# B&R Automation Studio project ARuser
Automation Studio 6.1.1.14; technology packages: mappView 6.1.1, OpcUaCs 6.0.0

## Configuration PC

CPU PC_any, AutomationRuntime 6.1.1, Build 11.3.0, Safety 0.0, Vc 

### Hardware
```
PC : PC_any v1.1.2.0 (OrderNumber=PC)
  Connector IF3:
    InaPort = 11159
  ConfigurationID = ARuser_PC
  VolatileGlobalPvSize = 200000
  Cyclic1Duration = 10000
  Cyclic3Tolerance = 60000000
  Cyclic8Duration = 10000
  FileDevice1
  FileDeviceName1 = FileDevice
  FileDevicePath1 = C:\Users\hendricksf\Desktop
  ActivateFtpServer = 1
  ActivateWebServer = 1
  ActivateSdm = 1
```

## Configuration X20CP

CPU X20CP3585, AutomationRuntime J4.93, Build 4.1.2, Vc V4.52.0

CPU X20CP3685, AutomationRuntime 6.1.1, Build 11.3.0, Vc 

### Hardware
```
X20CP3685 : X20CP3685 v1.8.1.0
  Connector IF2:
    ActivateDevice = 1
  Connector IF3:
    DNAConfiguration = manual
  ConfigurationID = ARuser_X20CP
  UserPartitionSize = 16
  VolatileGlobalPvSize = 120000
  FileDevice1
  FileDeviceName1 = USER
  FileDevicePath1 = USER_PATH
```

## Logical view

Binary libraries used (declarations not repeated): ArUser, MpUserX 5.24.3

### sys_lib.var
```iecst
(*error codes of the SYS_LIB services*)
VAR CONSTANT
	ERR_BUR_MO_NOTFOUND     	: UINT	:= 3019;    (*module not found*)
	ERR_BUR_ILLSTATE			: UINT	:= 3302;	(*illegal state of object*)
	ERR_BUR_ILLTYP				: UINT	:= 3311;	(*SYSreset - invalid input value for mode*)
	ERR_BUR_ILLPAR				: UINT	:= 3317;	(*illegal parameter*)
	ERR_BUR_ILLOBJ				: UINT	:= 3324;	(*object does not exist*)
	ERR_BUR_NOENTRY         	: UINT	:= 3332;    (*no entry*)
	ERR_BUR_TOOLONG_PVNAME		: UINT	:= 3333;	(*too long PV name*)
	ERR_BUR_ILLIDENT        	: UINT	:= 3336;    (*illegal ident*)
	ERR_BUR_NOTIME				: UINT	:= 3584;	(*time not available*)
	ERR_BUR_TMP_ALLOC			: UINT	:= 3601;	(*not enough continuous memory*)
	ERR_BUR_TMP_FREE			: UINT	:= 3701;	(*invalid pointer/length*)
END_VAR

(*state for object PLC task*)
VAR CONSTANT
	Z_ST_created				: UINT	:= 1;		(*object installed*)
	Z_ST_running				: UINT	:= 2;		(*object running*)
	Z_ST_blocked				: UINT	:= 3;		(*object stopped*)
	Z_ST_exist					: UINT	:= 16#00;	(*object exists*)
	Z_ST_installed				: UINT	:= 16#82;	(*temporary status during installation*)
	Z_ST_PVinstalled			: UINT	:= 16#83;	(*temporary status during installation*)
	Z_ST_IOinstalled			: UINT	:= 16#84;	(*temporary status during installation*)
	Z_ST_IOdeinstalled			: UINT	:= 16#85;	(*temporary status during installation*)
	Z_ST_PVdeinstalled			: UINT	:= 16#86;	(*temporary status during installation*)
	Z_ST_delete					: UINT	:= 16#87;	(*temporary status during installation*)
	Z_ST_stdebug				: UINT	:= 16#88;	(*temporary status during installation*)
	Z_ST_tmp_suspended			: UINT	:= 16#90;	(*object temporarily stopped*)
END_VAR

(*elementary data types*)
VAR CONSTANT
	SYSLIB_IEC_TYPE_USER_DEFINED	: USINT	:= 0;	(*User-defined data type*)
	SYSLIB_IEC_TYPE_USER_DEFINED_2	: USINT	:= 15;	(*User-defined data type (legacy: array of structs)*)
	SYSLIB_IEC_TYPE_BOOL			: USINT	:= 1;	(*8 Bit containing a boolean value FALSE=0 or TRUE=1*)
	SYSLIB_IEC_TYPE_SINT			: USINT	:= 2;	(*8 Bit signed integer*)
	SYSLIB_IEC_TYPE_INT				: USINT	:= 3;	(*16 Bit signed integer*)
	SYSLIB_IEC_TYPE_DINT			: USINT	:= 4;	(*32 Bit signed integer*)
	SYSLIB_IEC_TYPE_USINT			: USINT	:= 5;	(*8 Bit unsigned integer*)
	SYSLIB_IEC_TYPE_UINT			: USINT	:= 6;	(*16 Bit unsigned integer*)
	SYSLIB_IEC_TYPE_UDINT			: USINT	:= 7;	(*32 Bit unsigned integer*)
	SYSLIB_IEC_TYPE_REAL			: USINT	:= 8;	(*32 Bit floating point number*)
	SYSLIB_IEC_TYPE_STRING			: USINT	:= 9;	(*Variable-length single-byte character string*)
	SYSLIB_IEC_TYPE_DATE_AND_TIME	: USINT	:= 11;	(*32 Bit of Date in Seconds since 01.01.1970 00:00:00*)
	SYSLIB_IEC_TYPE_TIME			: USINT	:= 12;	(*32 Bit of Time in ms*)
	SYSLIB_IEC_TYPE_DATE			: USINT	:= 13;	(*32 Bit of Date (only)*)
	SYSLIB_IEC_TYPE_LREAL			: USINT	:= 14;	(*64 Bit floating point number*)
	SYSLIB_IEC_TYPE_TIME_OF_DAY		: USINT	:= 16;	(*32 Bit Time of day (only)*)
	SYSLIB_IEC_TYPE_BYTE			: USINT	:= 17;	(*Bit string of length 8*)
	SYSLIB_IEC_TYPE_WORD			: USINT	:= 18;	(*Bit string of length 16*)
	SYSLIB_IEC_TYPE_DWORD			: USINT	:= 19;	(*Bit string of length 32*)
	SYSLIB_IEC_TYPE_WSTRING			: USINT	:= 21;	(*Variable-length double-byte character string*)
END_VAR

(*shutdown/reboot types*)
VAR CONSTANT
	SYSLIB_WARMSTART				: USINT	:= 16#01;	(*WARMSTART (with restart)*)
	SYSLIB_COLDSTART				: USINT	:= 16#02;	(*COLDSTART (with restart)*)
	SYSLIB_WARMSTART_NO_REBOOT		: USINT	:= 16#11;	(*WARMSTART (no restart, only shutdown)*)
	SYSLIB_COLDSTART_NO_REBOOT		: USINT	:= 16#12;	(*COLDSTART (no restart, only shutdown)*)
	SYSLIB_DIAGNOSTICS				: USINT	:= 16#20;	(*DIAGNOSTICS (with restart)*)
	SYSLIB_SERVICE					: USINT	:= 16#40;	(*SERVICE (with restart) *)
END_VAR
```

### UserVariables.var
```iecst
(*Global constants*)
VAR CONSTANT
	MAX_USER_ROLES : USINT := 20; (*Maximum number of user roles*)
	MAX_USER_NAMES : USINT := 50; (*Maximum number of users*)
	MAX_USER_CLIENTS : USINT := 2; (*Maximum number of concurrent web clients*)
	MAX_USER_ITEM_LEN : USINT := 60; (*String length for users and roles*)
END_VAR
VAR
	DEFAULT_ROLE : STRING[80] := 'Everyone'; (*Default role when user was created*)
END_VAR
(*Global variable structure*)
VAR
	ArUser : userMAIN; (*Type for user data management*)
	RFID : rfidMAIN;
END_VAR
```

### changelog.txt
```
Version 1.2
- Update project to AS6
- Workaround for user create not assigning default role

Version 1.1
- Dont disable enable button in RFID group
- Added user partition for export/import
- Fixed export path not connected to ArUser.PAR.FilePath in mappView

Version 1.0
- Fixed password is not created

Version 0.8
- Update user management to version 0.8
- Added support for RFID reader 5E9030

Version 0.7
- Clear password field when user is created, password is changed, login or logout
- Removed user anonymous from user list
- Increased length of status message

Version 0.6
- Added message box before deleting user
- Changed constant to avoid conflict with other samples
- Fixed user selection after create and rename
- Updated mappView to 5.7.1
- Code optimizations

Version 0.5
- Code cleanup

Version 0.5
- Multi client support
- Changed error structure

Version 0.4
- Software structure change to work with future expansion
- Make sure passwords match before user is created
- Added support for RFID reader

Version 0.3
- Automatically set password when new user is created
- Erase password field when user logs out
- New command to rename user

Version 0.2
- Make sure last user can not be deleted
- Make sure last user can not delete himself
- Make sure last user can not be deleted
- Added group box with login
- Added message boxes for success and failed commands
- Visual tweaks and bugfixes

Version 0.1
- First public release
```

### Program Logical/mappUser/UserManagement

#### Variables.var
```iecst
(*General*)
VAR
	UserManagementState : userManagementEnum := IdleUser; (*State Machine for UserManagementState*)
	ArUserCreate_0 : ArUserCreate; (*Create an user with given name; default no password *)
	ArUserDelete_0 : ArUserDelete; (*Delete an user  *)
	ArUserExport_0 : ArUserExportEx; (*Export all user and role data*)
	ArUserImport_0 : ArUserImportEx; (*Import all user and role data*)
	ArUserSetPassword_0 : ArUserSetPassword; (*Set user password*)
	ArUserAssignRole_0 : ArUserAssignRole; (*Aisign a role to a user*)
	ArUserReleaseRole_0 : ArUserReleaseRole; (*Remove a role from a user*)
	ArUserGetNext_0 : ArUserGetNext; (*Get next user information*)
	ArUserGetFirst_0 : ArUserGetFirst; (*Get first user information*)
	ArUserInitList_0 : ArUserInitList; (*Initialize user or role list*)
	ArUserDestroyList_0 : ArUserDestroyList; (*Free up memory for list*)
	ArUserIdent : ArUserIdentType; (*Ident from user ot role list*)
	ArUserGetProperty_0 : ArUserGetProperty; (*Read property*)
	ArUserSetProperty_0 : ArUserSetProperty; (*Write a property*)
	PropertyName : STRING[100]; (*Name of the property*)
	tmpUserIdx : USINT;
	tmpUser : STRING[MAX_USER_ITEM_LEN];
	tmpUserOld : STRING[MAX_USER_ITEM_LEN];
	tmpUserNew : STRING[MAX_USER_ITEM_LEN];
	idx : USINT;
	idy : USINT;
	override : USINT;
END_VAR
VAR CONSTANT
	MAX_CYCLES : USINT := 10; (*Maximum number of override cycles*)
END_VAR
(*Loop counter*)
VAR
	RoleCounter : USINT;
	UserCounter : USINT;
	UserCounterTotal : ARRAY[0..MAX_USER_CLIENTS] OF USINT;
END_VAR
(*List types *)
VAR CONSTANT
	USER_LISTTYPE : BYTE := 1; (*List Type User*)
	ROLE_LISTTYPE : BYTE := 2; (*List Type Role*)
	USERROLE_LISTTYPE : BYTE := 3; (*List Type UserRole*)
END_VAR
(*Error Constants*)
VAR CONSTANT
	ERR_PASSWORD_MISMATCH : DINT := 50000; (*Passwords dont match*)
	ERR_USER_LIST_TOO_SHORT : DINT := 50001; (*More users found than fit into user list*)
	ERR_ROLE_LIST_TOO_SHORT : DINT := 50002; (*More roles found than fit into the role list*)
	ERR_DELETE_CURRENT_USER : DINT := 50003; (*Logged in user can not be deleted*)
	ERR_RENAME_CURRENT_USER : DINT := 50004; (*Logged in user can not be renamed*)
	ERR_USER_ROLE_NAME_SIZE : DINT := 50005; (*Logged in user can not be renamed*)
	ERR_USER_TOO_MANY_CLIENTS : DINT := 50010; (*More than 3 clients try to connect to user managment*)
	END_OF_LIST : DINT := -2144327714; (*End of list reached*)
	ONE : BOOL := TRUE;
END_VAR
```

#### Main.st
```iecst
// --------------------------------------------------------------------------------------------------------------------
// General user task. This is a support task for the mappView visualization. The following functions are implemneted
// - Create,rename and delete user
// - Create and delete roles
// - Change password and assign roles to users
// - Export and import user data
// Version 0.8
// --------------------------------------------------------------------------------------------------------------------
PROGRAM _INIT
	ArUser.CMD.ListRefresh	:= TRUE;								// Refresh user data on boot
END_PROGRAM

PROGRAM _CYCLIC

	FOR override:=0 TO MAX_CYCLES DO
		// --------------------------------------------------------------------------------------------------------------------
		// User managment state machine
		// --------------------------------------------------------------------------------------------------------------------
		CASE UserManagementState OF
			// --------------------------------------------------------------------------------------------------------------------
			// Wait for new command
			// --------------------------------------------------------------------------------------------------------------------
			IdleUser:
				// --------------------------------------------------------------------------------------------------------------------
				// Make sure we dont exceed maximum number of web clients
				IF(ArUser.PAR.VisuSlotID >= SIZEOF(ArUser.VIS)/SIZEOF(ArUser.VIS[0])) THEN
					ArUser.ERR.No := ERR_USER_TOO_MANY_CLIENTS;
					ArUser.ERR.State := UserManagementState;
					UserManagementState := ErrorUser;
					RETURN;
				END_IF

				// --------------------------------------------------------------------------------------------------------------------
				// Some general UI tasks
				FOR idy:=0 TO SIZEOF(ArUser.VIS)/SIZEOF(ArUser.VIS[0])-1 DO
					// --------------------------------------------------------------------------------------------------------------------
					// Create role list for current user
					idx := 0;
					brsmemset(ADR(ArUser.VIS[idy].ListUserRole), 0, SIZEOF(ArUser.VIS[idy].ListUserRole));
					WHILE brsstrcmp(ADR(ArUser.DAT.Users[ArUser.VIS[idy].ListUserIndex].Roles[idx]), ADR('')) <> 0 DO
						String2DataProvider(ADR(ArUser.DAT.Users[ArUser.VIS[idy].ListUserIndex].Roles[idx]), ADR(ArUser.VIS[idy].ListUserRole[idx]));
						idx := idx + 1;
					END_WHILE;
					// Make sure we dont delete last user role
					IF(idx > 1) THEN
						ArUser.VIS[idy].RoleDeleteEnabled := TRUE;
					ELSE
						ArUser.VIS[idy].RoleDeleteEnabled := FALSE;
					END_IF
					// Make sure we dont delete last user
					IF(UserCounterTotal[idy] > 0) THEN
						ArUser.VIS[idy].UserDeleteEnabled := TRUE;
					ELSE
						ArUser.VIS[idy].UserDeleteEnabled := FALSE;
					END_IF
				END_FOR;

				// --------------------------------------------------------------------------------------------------------------------
				// Create new user
				IF  (ArUser.CMD.UserCreate) THEN
					// Make sure passwords match before user is created
					IF((ArUser.PAR.Password <> '' OR ArUser.PAR.PasswordRepeat <> '') AND ArUser.PAR.Password <> ArUser.PAR.PasswordRepeat) THEN
						ArUser.ERR.No := ERR_PASSWORD_MISMATCH;
						ArUser.ERR.State := UserManagementState;
						UserManagementState := ErrorUser;
					ELSE
						tmpUser := ArUser.PAR.UserName;
						ArUserCreate_0(Execute := FALSE);
						ArUserSetPassword_0(Execute := FALSE);
						UserManagementState := CreateUser;
					END_IF
				// Assign role to user
				ELSIF (ArUser.CMD.RoleAssign) THEN
					tmpUser := ArUser.PAR.UserName;
					ArUserAssignRole_0(Execute := FALSE);
					ArUser.PAR.UserRole := ArUser.DAT.Roles[ArUser.VIS[ArUser.PAR.VisuSlotID].ListRoleIndex];
					UserManagementState := AssignRole;
				// Remove role from user
				ELSIF (ArUser.CMD.RoleRemove) THEN
					tmpUser := ArUser.PAR.UserName;
					ArUserReleaseRole_0(Execute := FALSE);
					ArUser.PAR.UserRole := ArUser.DAT.Users[ArUser.VIS[ArUser.PAR.VisuSlotID].ListUserIndex].Roles[ArUser.VIS[ArUser.PAR.VisuSlotID].ListUserRoleIndex];
					UserManagementState := ReleaseRole;
				// Delete user
				ELSIF (ArUser.CMD.UserDelete) THEN
					// Make sure we dont delete user that is logged in
					IF(brsstrcmp(ADR(ArUser.DAT.UserActive[ArUser.PAR.VisuSlotID]), ADR(ArUser.PAR.UserName)) = 0) THEN
						ArUser.ERR.No := ERR_DELETE_CURRENT_USER;
						ArUser.ERR.State := UserManagementState;
						UserManagementState := ErrorUser;
					ELSE
						tmpUser := ArUser.PAR.UserName;
						ArUserDelete_0(Execute := FALSE);
						UserManagementState := DeleteUser;
					END_IF
				// Rename user
				ELSIF (ArUser.CMD.UserRename) THEN
					// Make sure we dont delete user that is logged in
					IF(brsstrcmp(ADR(ArUser.DAT.UserActive[ArUser.PAR.VisuSlotID]), ADR(ArUser.PAR.UserName)) = 0) THEN
						ArUser.ERR.No := ERR_RENAME_CURRENT_USER;
						ArUser.ERR.State := UserManagementState;
						UserManagementState := ErrorUser;
					ELSE
						tmpUserOld := ArUser.PAR.UserName;
						tmpUser := ArUser.PAR.UserNameNew;
						ArUserGetProperty_0(Execute := FALSE);
						ArUserSetProperty_0(Execute := FALSE);
						ArUserAssignRole_0(Execute := FALSE);
						ArUserDelete_0(Execute := FALSE);
						UserManagementState := RenameUser;
					END_IF
				// Export user data
				ELSIF (ArUser.CMD.Export) THEN
					ArUserExport_0(Execute := FALSE);
					UserManagementState := ExportList;
				// Import user data
				ELSIF (ArUser.CMD.Import) THEN
					ArUserImport_0(Execute := FALSE);
					UserManagementState := ImportList;
				// Change user password
				ELSIF (ArUser.CMD.PasswordChange) THEN
					tmpUser := ArUser.PAR.UserName;
					ArUserSetPassword_0(Execute := FALSE);
					UserManagementState := ComparePassword;
				// Refresh user list
				ELSIF (ArUser.CMD.ListRefresh) THEN
					tmpUser := '';
					UserManagementState := CreateUserListGetFirst;
				END_IF;

				// --------------------------------------------------------------------------------------------------------------------
				// Reset fields on new command
				FOR idx:=0 TO SIZEOF(ArUser.CMD) DO
					IF brsmemcmp(ADR(ArUser.CMD) + idx, ADR(ONE), 1) = 0 THEN
						ArUser.DAT.Status := '';
	 				END_IF
				END_FOR
				ArUser.CMD.ErrorReset := FALSE;

				// Abot override when no command is active
				IF (UserManagementState = IdleUser) THEN
					RETURN;
				END_IF
			// --------------------------------------------------------------------------------------------------------------------
			// Create new user
			// --------------------------------------------------------------------------------------------------------------------
			CreateUser:
				ArUserCreate_0(Execute := TRUE , UserName := tmpUser);

				// --------------------------------------------------------------------------------------------------------------------
				// Success
				IF ArUserCreate_0.Done AND NOT ArUserCreate_0.Busy THEN
					// Create new user
					IF(ArUser.CMD.UserCreate) THEN
						// --------------------------------------------------------------------------------------------------------------------
						// Success
						ArUserAssignRole_0(Execute := TRUE, UserName := tmpUser, RoleName := DEFAULT_ROLE);
						ArUserAssignRole_0(Execute := TRUE, UserName := tmpUser, RoleName := DEFAULT_ROLE);
						IF ArUserAssignRole_0.Done AND NOT ArUserAssignRole_0.Busy THEN
							ArUserAssignRole_0(Execute := FALSE);

							ArUser.DAT.Status := 'User ';
							brsstrcat(ADR(ArUser.DAT.Status), ADR(tmpUser));
							brsstrcat(ADR(ArUser.DAT.Status), ADR(' created'));
							// Set password when it exists
							IF ArUser.PAR.Password <> '' THEN
								UserManagementState := ComparePassword;
							ELSE
								ArUser.PAR.UserName := '';
								UserManagementState := CreateUserListGetFirst;
							END_IF;

							RETURN;
							// Error
						ELSIF ArUserAssignRole_0.Error THEN
							ArUser.ERR.No := ArUserAssignRole_0.ErrorID;
							ArUser.ERR.State := UserManagementState;
							UserManagementState := ErrorUser;
						END_IF
						// Rename existing user
					ELSE
						PropertyName := 'UserID';
						UserManagementState := PropertyRead;
					END_IF
					// Error
				ELSIF ArUserCreate_0.Error THEN
					ArUser.ERR.No := ArUserCreate_0.ErrorID;
					ArUser.ERR.State := UserManagementState;
					UserManagementState := ErrorUser;
				END_IF;

			// --------------------------------------------------------------------------------------------------------------------
			// Assign user role
			// --------------------------------------------------------------------------------------------------------------------
			AssignRole:
				ArUserAssignRole_0(Execute := TRUE, UserName := tmpUser, RoleName := ArUser.PAR.UserRole);

				// --------------------------------------------------------------------------------------------------------------------
				// Success
				IF ArUser.CMD.RoleAssign AND ArUserAssignRole_0.Done AND NOT ArUserAssignRole_0.Busy THEN
					ArUser.DAT.Status := 'Role >';
					brsstrcat(ADR(ArUser.DAT.Status), ADR(ArUser.PAR.UserRole));
					brsstrcat(ADR(ArUser.DAT.Status), ADR('< assigned to user '));
					brsstrcat(ADR(ArUser.DAT.Status), ADR(tmpUser));
					ArUser.PAR.UserName := '';
					UserManagementState := CreateUserListGetFirst;
				ELSIF ArUser.CMD.UserRename AND ((ArUserAssignRole_0.Done AND NOT ArUserAssignRole_0.Busy) OR (ArUserAssignRole_0.ErrorID = arUSER_ERR_ALREADY_EXISTS)) THEN
					idx := idx +1;
					// Assign next role if it exists
					IF ArUser.DAT.Users[tmpUserIdx].Roles[idx] <> '' AND idx < MAX_USER_ROLES THEN
						ArUserAssignRole_0(Execute := FALSE);
						ArUser.PAR.UserRole := ArUser.DAT.Users[tmpUserIdx].Roles[idx];
					// Delete old user
					ELSE
						// Move user names around
						tmpUserNew 	:= tmpUser;
						tmpUser 	:= tmpUserOld;
						UserManagementState := DeleteUser;
					END_IF
				// Error
				ELSIF ArUserAssignRole_0.Error THEN
					ArUser.ERR.No := ArUserAssignRole_0.ErrorID;
					ArUser.ERR.State := UserManagementState;
					UserManagementState := ErrorUser;
				END_IF;

			// --------------------------------------------------------------------------------------------------------------------
			// Release user role
			// --------------------------------------------------------------------------------------------------------------------
			ReleaseRole:
				ArUserReleaseRole_0(Execute := TRUE, UserName := tmpUser, RoleName := ArUser.PAR.UserRole);

				// --------------------------------------------------------------------------------------------------------------------
				// Success
				IF ArUserReleaseRole_0.Done AND NOT ArUserReleaseRole_0.Busy THEN
					ArUser.DAT.Status := 'Role >';
					brsstrcat(ADR(ArUser.DAT.Status), ADR(ArUser.PAR.UserRole));
					brsstrcat(ADR(ArUser.DAT.Status), ADR('< removed from user '));
					brsstrcat(ADR(ArUser.DAT.Status), ADR(tmpUser));
					ArUser.PAR.UserName := '';
					UserManagementState := CreateUserListGetFirst;
				// Error
				ELSIF ArUserReleaseRole_0.Error THEN
					ArUser.ERR.No := ArUserReleaseRole_0.ErrorID;
					ArUser.ERR.State := UserManagementState;
					UserManagementState := ErrorUser;
				END_IF;

			// --------------------------------------------------------------------------------------------------------------------
			// Delete user
			// --------------------------------------------------------------------------------------------------------------------
			DeleteUser:
				ArUserDelete_0(Execute := TRUE, UserName := tmpUser);

				// --------------------------------------------------------------------------------------------------------------------
				// Success
				IF ArUserDelete_0.Done AND NOT ArUserDelete_0.Busy THEN
					// User delete command
					IF ArUser.CMD.UserDelete THEN
						ArUser.DAT.Status := 'User >';
						brsstrcat(ADR(ArUser.DAT.Status), ADR(tmpUser));
						brsstrcat(ADR(ArUser.DAT.Status), ADR('< deleted'));
						// User rename command
					ELSE
						ArUser.DAT.Status := 'User ';
						brsstrcat(ADR(ArUser.DAT.Status), ADR(tmpUserOld));
						brsstrcat(ADR(ArUser.DAT.Status), ADR(' renamed to >'));
						brsstrcat(ADR(ArUser.DAT.Status), ADR(ArUser.PAR.UserNameNew));
						brsstrcat(ADR(ArUser.DAT.Status), ADR('<'));
					END_IF
					ArUser.PAR.UserName := '';
					tmpUser := '';
					UserManagementState := CreateUserListGetFirst;
				// Error
				ELSIF ArUserDelete_0.Error THEN
					ArUser.ERR.No := ArUserDelete_0.ErrorID;
					ArUser.ERR.State := UserManagementState;
					UserManagementState := ErrorUser;
				END_IF;

			// --------------------------------------------------------------------------------------------------------------------
			// Rename user
			// --------------------------------------------------------------------------------------------------------------------
			RenameUser:
				tmpUserIdx := 0;
				// Find user name in list
				WHILE (brsstrcmp(ADR(ArUser.DAT.Users[tmpUserIdx].Name), ADR(tmpUserOld)) <> 0) AND (tmpUserIdx < MAX_USER_NAMES) DO
					tmpUserIdx := tmpUserIdx + 1;
				END_WHILE;

				// --------------------------------------------------------------------------------------------------------------------
				// Success
				IF(tmpUserIdx < MAX_USER_NAMES) THEN
					ArUserCreate_0(Execute := FALSE);
					UserManagementState := CreateUser;
				// Error when user was not found
				ELSE
					ArUser.ERR.No := arUSER_ERR_DOES_NOT_EXIST;
					ArUser.ERR.State := UserManagementState;
					UserManagementState := ErrorUser;
				END_IF

			// --------------------------------------------------------------------------------------------------------------------
			// Read user property
			// --------------------------------------------------------------------------------------------------------------------
			PropertyRead:
				ArUserGetProperty_0(Execute := TRUE, ElementType := arUSER_USER_PROPERTIES, ElementName := tmpUserOld, PropertyName := PropertyName);

				// --------------------------------------------------------------------------------------------------------------------
				// Success
				IF ArUserGetProperty_0.Done AND NOT ArUserGetProperty_0.Busy THEN
					ArUserSetProperty_0(Execute := FALSE);
					UserManagementState := PropertyWrite;
				// Error
				ELSIF ArUserGetProperty_0.Error THEN
					ArUser.ERR.No := ArUserGetProperty_0.ErrorID;
					ArUser.ERR.State := UserManagementState;
					UserManagementState := ErrorUser;
				END_IF;
			// --------------------------------------------------------------------------------------------------------------------
			// Write user property
			// --------------------------------------------------------------------------------------------------------------------
			PropertyWrite:
				ArUserSetProperty_0(Execute := TRUE, ElementType := arUSER_USER_PROPERTIES, ElementName := tmpUser, PropertyName := PropertyName, PropertyValue := ArUserGetProperty_0.PropertyValue);

				// --------------------------------------------------------------------------------------------------------------------
				// Success
				IF ArUserSetProperty_0.Done AND NOT ArUserSetProperty_0.Busy THEN
					// Read password after user ID
					IF PropertyName = 'UserID' THEN
						PropertyName := 'Password';
						ArUserGetProperty_0(Execute := FALSE);
						UserManagementState := PropertyRead;
						// Assign roles after password
					ELSIF PropertyName = 'Password' THEN
						idx := 0;
						ArUser.PAR.UserRole := ArUser.DAT.Users[tmpUserIdx].Roles[idx];
						UserManagementState := AssignRole;
					END_IF
				// Error
				ELSIF ArUserSetProperty_0.Error THEN
					ArUser.ERR.No := ArUserSetProperty_0.ErrorID;
					ArUser.ERR.State := UserManagementState;
					UserManagementState := ErrorUser;
				END_IF;

			// --------------------------------------------------------------------------------------------------------------------
			// Export user list to file
			// --------------------------------------------------------------------------------------------------------------------
			ExportList:
				ArUserExport_0(Execute := TRUE , LocalPath := ArUser.PAR.FilePath);

				// --------------------------------------------------------------------------------------------------------------------
				// Success
				IF ArUserExport_0.Done AND NOT ArUserExport_0.Busy THEN
					ArUser.DAT.Status := 'Export finished';
					ArUser.CMD.Export := FALSE;
					ArUser.VIS[ArUser.PAR.VisuSlotID].ShowMessageBoxOK := TRUE;
					UserManagementState := IdleUser;
					RETURN;
				// Error
				ELSIF ArUserExport_0.Error THEN
					ArUser.ERR.No := ArUserExport_0.ErrorID;
					ArUser.ERR.State := UserManagementState;
					UserManagementState := ErrorUser;
				END_IF;

			// --------------------------------------------------------------------------------------------------------------------
			// Import user list from file
			// --------------------------------------------------------------------------------------------------------------------
			ImportList:
				ArUserImport_0(Execute := TRUE , LocalPath := ArUser.PAR.FilePath);

				// --------------------------------------------------------------------------------------------------------------------
				// Success
				IF ArUserImport_0.Done AND NOT ArUserImport_0.Busy THEN
					ArUser.DAT.Status := 'Import finished';
					ArUser.CMD.Import := FALSE;
					ArUser.VIS[ArUser.PAR.VisuSlotID].ShowMessageBoxOK := TRUE;
					UserManagementState := CreateUserListGetFirst;
				// Error
				ELSIF ArUserImport_0.Error THEN
					ArUser.ERR.No := ArUserImport_0.ErrorID;
					ArUser.ERR.State := UserManagementState;
					UserManagementState := ErrorUser;
				END_IF;

			// --------------------------------------------------------------------------------------------------------------------
			// Change password, make sure both passwords are correct
			// --------------------------------------------------------------------------------------------------------------------
			ComparePassword:
				// --------------------------------------------------------------------------------------------------------------------
				// Success
				IF brsstrcmp(ADR(ArUser.PAR.Password), ADR(ArUser.PAR.PasswordRepeat)) = 0 THEN
					UserManagementState := ChangePassword;
				// Error
				ELSE
					ArUser.ERR.No := ERR_PASSWORD_MISMATCH;
					ArUser.ERR.State := UserManagementState;
					UserManagementState := ErrorUser;
				END_IF;

			// --------------------------------------------------------------------------------------------------------------------
			// Change password, execute password change
			// --------------------------------------------------------------------------------------------------------------------
			ChangePassword:
				ArUserSetPassword_0(Execute := TRUE, UserName := tmpUser, Password := ArUser.PAR.Password);

				// --------------------------------------------------------------------------------------------------------------------
				// Success
				IF ArUserSetPassword_0.Done AND NOT ArUserSetPassword_0.Busy THEN
					IF ArUser.CMD.PasswordChange THEN
						ArUser.DAT.Status := 'Password for user >';
						brsstrcat(ADR(ArUser.DAT.Status), ADR(tmpUser));
						brsstrcat(ADR(ArUser.DAT.Status), ADR('< changed'));
						ArUser.PAR.Password := '';
						ArUser.PAR.PasswordRepeat := '';
						ArUser.CMD.PasswordChange := FALSE;
						ArUser.VIS[ArUser.PAR.VisuSlotID].ShowMessageBoxOK := TRUE;
						UserManagementState := IdleUser;
						RETURN;
					ELSE
						UserManagementState := CreateUserListGetFirst;
					END_IF;
				// Error
				ELSIF ArUserSetPassword_0.Error THEN
					ArUser.ERR.No := ArUserSetPassword_0.ErrorID;
					ArUser.ERR.State := UserManagementState;
					UserManagementState := ErrorUser;
				END_IF;

			// --------------------------------------------------------------------------------------------------------------------
			// Create list of users and roles
			// --------------------------------------------------------------------------------------------------------------------
			CreateUserListGetFirst:
				// Initialize user list
				ArUserInitList_0(Execute := TRUE, ListType := USER_LISTTYPE, ElementName :='');

				// --------------------------------------------------------------------------------------------------------------------
				// Get first user name
				IF ArUserInitList_0.Done AND NOT ArUserInitList_0.Busy THEN
					ArUserGetFirst_0(Execute := TRUE , List := ArUserInitList_0.List );

					// --------------------------------------------------------------------------------------------------------------------
					// Success
					IF ArUserGetFirst_0.Done THEN
						// Clear data, store user name and generate data provider for vis
						brsmemset(ADR(ArUser.DAT.Users), 0, SIZEOF(ArUser.DAT.Users));
						brsmemset(ADR(ArUser.VIS[ArUser.PAR.VisuSlotID].ListUsers), 0, SIZEOF(ArUser.VIS[ArUser.PAR.VisuSlotID].ListUsers));
						brsmemset(ADR(ArUser.VIS[ArUser.PAR.VisuSlotID].ListRoles), 0, SIZEOF(ArUser.VIS[ArUser.PAR.VisuSlotID].ListRoles));
						UserCounter := 0;

						// Make sure user name fits
						IF(brsstrlen(ADR(ArUserGetFirst_0.ElementName)) < MAX_USER_ITEM_LEN) THEN
							// Ignore use an anonymous
							IF(ArUserGetFirst_0.ElementName <> 'Anonymous') THEN
								ArUser.DAT.Users[UserCounter].Name := ArUserGetFirst_0.ElementName;
								String2DataProvider(ADR(ArUserGetFirst_0.ElementName), ADR(ArUser.VIS[ArUser.PAR.VisuSlotID].ListUsers[UserCounter]));
								UserCounter := 1;
							ELSE
								UserCounter := 0;
							END_IF
							// Reset function block and init counters
							ArUserGetFirst_0(Execute := FALSE);
							RoleCounter := 0;
							UserManagementState := CreateUserListGetNext;
						// User name is too long
						ELSE
							ArUser.ERR.No := ERR_USER_ROLE_NAME_SIZE;
							ArUser.ERR.State := UserManagementState;
							UserManagementState := ErrorUser;
						END_IF;
					// Error
					ELSIF ArUserGetFirst_0.Error THEN
						ArUser.ERR.No := ArUserGetFirst_0.ErrorID;
						ArUser.ERR.State := UserManagementState;
						UserManagementState := ErrorUser;
					END_IF;
				// Error
				ELSIF ArUserInitList_0.Error THEN
					ArUser.ERR.No := ArUserInitList_0.ErrorID;
					ArUser.ERR.State := UserManagementState;
					UserManagementState := ErrorUser;
				END_IF;

			CreateUserListGetNext:
				// Make sure we have space left
				IF UserCounter < SIZEOF(ArUser.DAT.Users)/SIZEOF(ArUser.DAT.Users[0]) THEN
					// Get next user
					ArUserGetNext_0(Execute := TRUE , List := ArUserInitList_0.List);

					// --------------------------------------------------------------------------------------------------------------------
					// Success
					IF ArUserGetNext_0.Done THEN
						// Make sure user name fits
						IF(brsstrlen(ADR(ArUserGetNext_0.ElementName)) < MAX_USER_ITEM_LEN) THEN
							// Ignore use an anonymous
							IF(ArUserGetNext_0.ElementName <> 'Anonymous') THEN
								// Store user name and generate data provider for vis
								ArUser.DAT.Users[UserCounter].Name := ArUserGetNext_0.ElementName;
								String2DataProvider(ADR(ArUserGetNext_0.ElementName), ADR(ArUser.VIS[ArUser.PAR.VisuSlotID].ListUsers[UserCounter]));
								// Reset function block and get next name
								UserCounter := UserCounter + 1;
							END_IF
							ArUserGetNext_0(Execute := FALSE);
						// User name is too long
						ELSE
							ArUser.ERR.No := ERR_USER_ROLE_NAME_SIZE;
							ArUser.ERR.State := UserManagementState;
							UserManagementState := ErrorUser;
						END_IF;
					// Error
					ELSIF ArUserGetNext_0.Error AND NOT (ArUserGetNext_0.ErrorID = END_OF_LIST) THEN
						ArUser.ERR.No := ArUserGetNext_0.ErrorID;
						ArUser.ERR.State := UserManagementState;
						UserManagementState := ErrorUser;
					// List is complete
					ELSIF ArUserGetNext_0.ErrorID = END_OF_LIST THEN
						// Free up memory
						ArUserIdent := ArUserInitList_0.List;
						ArUserDestroyList_0(Execute := TRUE, List := ArUserIdent);
						ArUserDestroyList_0(Execute := FALSE, List := ArUserIdent);
						// Reset function blocks and counters
						ArUserGetNext_0(Execute := FALSE);
						ArUserGetFirst_0(Execute := FALSE);
						ArUserInitList_0(Execute := FALSE);
						UserCounterTotal[ArUser.PAR.VisuSlotID] := UserCounter;
						UserCounter := 0;
						RoleCounter := 0;
						UserManagementState := RoleListInitList;
					END_IF;
				// User list is too short
				ELSE
					ArUser.ERR.No := ERR_USER_LIST_TOO_SHORT;
					ArUser.ERR.State := UserManagementState;
					UserManagementState := ErrorUser;
				END_IF;

			// --------------------------------------------------------------------------------------------------------------------
			// Create table of roles assigned to the table of users
			// --------------------------------------------------------------------------------------------------------------------
			RoleListInitList:
				IF ArUser.DAT.Users[UserCounter].Name <> '' THEN
					ArUserInitList_0(Execute := TRUE, ListType := USERROLE_LISTTYPE , ElementName := ArUser.DAT.Users[UserCounter].Name);

					// --------------------------------------------------------------------------------------------------------------------
					// Success
					IF ArUserInitList_0.Done  AND NOT ArUserInitList_0.Busy THEN
						ArUserGetFirst_0(Execute := TRUE , List := ArUserInitList_0.List);
						// --------------------------------------------------------------------------------------------------------------------
						// Success
						IF ArUserGetFirst_0.Done THEN
							// Make sure role name fits
							IF(brsstrlen(ADR(ArUserInitList_0.ElementName)) < MAX_USER_ITEM_LEN) THEN
								ArUser.DAT.Users[UserCounter].Roles[0] := ArUserGetFirst_0.ElementName;
								ArUserGetFirst_0(Execute := FALSE , List := ArUserInitList_0.List);
								RoleCounter := 1;
								UserManagementState:= RoleListGetNext;
								// User role is too long
							ELSE
								ArUser.ERR.No := ERR_USER_ROLE_NAME_SIZE;
								ArUser.ERR.State := UserManagementState;
								UserManagementState := ErrorUser;
							END_IF;
						// Error
						ELSIF ArUserGetFirst_0.Error THEN
							ArUser.ERR.No := ArUserGetFirst_0.ErrorID;
							ArUser.ERR.State := UserManagementState;
							UserManagementState := ErrorUser;
						END_IF;
					// Error
					ELSIF ArUserInitList_0.Error THEN
						ArUser.ERR.No := ArUserInitList_0.ErrorID;
						ArUser.ERR.State := UserManagementState;
						UserManagementState := ErrorUser;
					END_IF;
				// Finish when user roles are complete
				ELSE
					// Reset function blocks
					ArUserInitList_0(Execute := FALSE);
					ArUserGetFirst_0(Execute := FALSE);
					UserCounter := 1;
					RoleCounter := 0;
					UserManagementState := CreateRoleListGetFirst;
				END_IF;

			RoleListGetNext:
				ArUserGetNext_0(Execute := TRUE, List := ArUserInitList_0.List);

				// --------------------------------------------------------------------------------------------------------------------
				// Success
				IF ArUserGetNext_0.Done THEN
					// Make sure user name fits
					IF(brsstrlen(ADR(ArUserGetNext_0.ElementName)) < MAX_USER_ITEM_LEN) THEN
						ArUser.DAT.Users[UserCounter].Roles[RoleCounter] := ArUserGetNext_0.ElementName;
						RoleCounter := RoleCounter + 1;
						ArUserGetNext_0(Execute := FALSE, List := ArUserInitList_0.List);
					// User role is too long
					ELSE
						ArUser.ERR.No := ERR_USER_ROLE_NAME_SIZE;
						ArUser.ERR.State := UserManagementState;
						UserManagementState := ErrorUser;
					END_IF;
				// List is complete
				ELSIF ArUserGetNext_0.ErrorID = END_OF_LIST THEN
					UserCounter := UserCounter + 1;
					// Free up memory
					ArUserIdent := ArUserInitList_0.List;
					ArUserDestroyList_0(Execute := TRUE, List := ArUserIdent);
					ArUserDestroyList_0(Execute := FALSE, List := ArUserIdent);
					// Reset function blocks
					ArUserGetNext_0(Execute := FALSE);
					ArUserInitList_0(Execute := FALSE);
					UserManagementState := RoleListInitList;
				// Error
				ELSIF ArUserGetNext_0.Error THEN
					ArUser.ERR.No := ArUserGetNext_0.ErrorID;
					ArUser.ERR.State := UserManagementState;
					UserManagementState := ErrorUser;
				END_IF;

			// --------------------------------------------------------------------------------------------------------------------
			// Create table of roles
			// --------------------------------------------------------------------------------------------------------------------
			CreateRoleListGetFirst:
				ArUserInitList_0(Execute := TRUE, ListType := ROLE_LISTTYPE , ElementName :='' );

				// --------------------------------------------------------------------------------------------------------------------
				// Success
				IF ArUserInitList_0.Done AND NOT ArUserInitList_0.Busy THEN
					ArUserGetFirst_0(Execute := TRUE , List := ArUserInitList_0.List );

					// --------------------------------------------------------------------------------------------------------------------
					// Store role names and generate data provider for vis
					IF ArUserGetFirst_0.Done THEN
						// Make sure role name fits
						IF(brsstrlen(ADR(ArUserGetFirst_0.ElementName)) < MAX_USER_ITEM_LEN) THEN
							ArUser.DAT.Roles[RoleCounter] := ArUserGetFirst_0.ElementName;
							String2DataProvider(ADR(ArUserGetFirst_0.ElementName), ADR(ArUser.VIS[ArUser.PAR.VisuSlotID].ListRoles[RoleCounter]));
							// Reset function block and init counters
							ArUserGetFirst_0(Execute := FALSE);
							RoleCounter := 1;
							UserManagementState := CreateRoleListGetNext;
							// Role name is too long
						ELSE
							ArUser.ERR.No := ERR_USER_ROLE_NAME_SIZE;
							ArUser.ERR.State := UserManagementState;
							UserManagementState := ErrorUser;
						END_IF;
					// Error
					ELSIF ArUserGetFirst_0.Error THEN
						ArUser.ERR.No := ArUserGetFirst_0.ErrorID;
						ArUser.ERR.State := UserManagementState;
						UserManagementState := ErrorUser;
					END_IF;
				// Error
				ELSIF ArUserInitList_0.Error THEN
					ArUser.ERR.No := ArUserInitList_0.ErrorID;
					ArUser.ERR.State := UserManagementState;
					UserManagementState := ErrorUser;
				END_IF;

			CreateRoleListGetNext:
				IF UserCounter < SIZEOF(ArUser.DAT.Roles)/SIZEOF(ArUser.DAT.Roles[0]) THEN
					ArUserGetNext_0(Execute := TRUE , List := ArUserInitList_0.List);

					// --------------------------------------------------------------------------------------------------------------------
					// Store user name and generate data provider for vis
					IF ArUserGetNext_0.Done THEN
						// Make sure user name fits
						IF(brsstrlen(ADR(ArUserGetNext_0.ElementName)) < MAX_USER_ITEM_LEN) THEN
							ArUser.DAT.Roles[RoleCounter] := ArUserGetNext_0.ElementName;
							String2DataProvider(ADR(ArUserGetNext_0.ElementName), ADR(ArUser.VIS[ArUser.PAR.VisuSlotID].ListRoles[RoleCounter]));
							// Reset function block and get next name
							RoleCounter := RoleCounter + 1;
							ArUserGetNext_0(Execute := FALSE);
						// Role name is too long
						ELSE
							ArUser.ERR.No := ERR_USER_ROLE_NAME_SIZE;
							ArUser.ERR.State := UserManagementState;
							UserManagementState := ErrorUser;
						END_IF;
					// Error
					ELSIF ArUserGetNext_0.Error AND NOT (ArUserGetNext_0.ErrorID = END_OF_LIST) THEN
						ArUser.ERR.No := ArUserGetNext_0.ErrorID;
						ArUser.ERR.State := UserManagementState;
						UserManagementState := ErrorUser;
					// End of list reached
					ELSIF ArUserGetNext_0.ErrorID = END_OF_LIST THEN
						// Show message box after succesful command except refresh
						IF(NOT ArUser.CMD.ListRefresh) THEN
							ArUser.VIS[ArUser.PAR.VisuSlotID].ShowMessageBoxOK := TRUE;
						END_IF
						// Reset function blocks
						ArUserGetNext_0(Execute := FALSE);
						ArUserInitList_0(Execute := FALSE);
						// Reset function blocks
						ArUserGetNext_0(Execute := FALSE);
						ArUserGetFirst_0(Execute := FALSE);
						ArUserInitList_0(Execute := FALSE);
						RoleCounter := 0;
						// Reset command
						brsmemset(ADR(ArUser.CMD), 0, SIZEOF(ArUser.CMD));
						// Select last user if possible
						IF(tmpUser <> '') THEN
							ArUser.VIS[ArUser.PAR.VisuSlotID].ListUserValue := tmpUser;
						ELSIF(tmpUserNew <> '') THEN
							ArUser.VIS[ArUser.PAR.VisuSlotID].ListUserValue := tmpUserNew;
						ELSE
							ArUser.PAR.UserName := ArUser.DAT.Users[0].Name;
						END_IF
						// Copy user data into all slots on first boot
						FOR idy:=0 TO SIZEOF(ArUser.VIS)/SIZEOF(ArUser.VIS[0])-1 DO
							IF(idy <> ArUser.PAR.VisuSlotID) THEN
								brsmemcpy(ADR(ArUser.VIS[idy].ListUsers), ADR(ArUser.VIS[ArUser.PAR.VisuSlotID].ListUsers), SIZEOF(ArUser.VIS[ArUser.PAR.VisuSlotID].ListUsers));
								brsmemcpy(ADR(ArUser.VIS[idy].ListRoles), ADR(ArUser.VIS[ArUser.PAR.VisuSlotID].ListRoles), SIZEOF(ArUser.VIS[ArUser.PAR.VisuSlotID].ListRoles));
								UserCounterTotal[idy] := UserCounterTotal[ArUser.PAR.VisuSlotID];
							END_IF
						END_FOR
						UserManagementState := IdleUser;
						RETURN;
					END_IF;
				// Role list is too short
				ELSE
					ArUser.ERR.No := ERR_ROLE_LIST_TOO_SHORT;
					ArUser.ERR.State := UserManagementState;
					UserManagementState := ErrorUser;
				END_IF;

			// --------------------------------------------------------------------------------------------------------------------
			// Error
			// --------------------------------------------------------------------------------------------------------------------
			ErrorUser:
				// --------------------------------------------------------------------------------------------------------------------
				// Reset function blocks
				ArUserInitList_0(Execute := FALSE);
				ArUserGetFirst_0(Execute := FALSE);
				ArUserGetNext_0(Execute := FALSE);
				ArUserCreate_0(Execute := FALSE);
				ArUserReleaseRole_0(Execute := FALSE);
				ArUserReleaseRole_0(Execute := FALSE);
				ArUserDelete_0(Execute := FALSE);
				ArUserGetProperty_0(Execute := FALSE);
				ArUserSetProperty_0(Execute := FALSE);
				ArUserSetPassword_0(Execute := FALSE);
				ArUserImport_0(Execute := FALSE);
				ArUserExport_0(Execute := FALSE);

				// --------------------------------------------------------------------------------------------------------------------
				// Generate text for most common errors
				IF(ArUser.ERR.No = arUSER_ERR_ALREADY_EXISTS) THEN
					ArUser.ERR.Text := 'ERR: User/Role already exists or is already assigned';
				ELSIF(ArUser.ERR.No = arUSER_ERR_PARAMETER) THEN
					ArUser.ERR.Text := 'ERR: User/Role is empty';
				ELSIF(ArUser.ERR.No = arUSER_ERR_DOES_NOT_EXIST) THEN
					ArUser.ERR.Text := 'ERR: User/Role does not exist';
				ELSIF(ArUser.ERR.No = ERR_PASSWORD_MISMATCH) THEN
					ArUser.ERR.Text := 'ERR: Passwords do not match';
				ELSIF(ArUser.ERR.No = ERR_USER_LIST_TOO_SHORT) THEN
					ArUser.ERR.Text := 'ERR: User list is too short';
				ELSIF(ArUser.ERR.No = ERR_ROLE_LIST_TOO_SHORT) THEN
					ArUser.ERR.Text := 'ERR: Role list is too short';
				ELSIF(ArUser.ERR.No = ERR_DELETE_CURRENT_USER) THEN
					ArUser.ERR.Text := 'ERR: Can not delete user that is logged in';
				ELSIF(ArUser.ERR.No = ERR_USER_ROLE_NAME_SIZE) THEN
					ArUser.ERR.Text := 'ERR: User name or role exceeds maximum size of ITEM_LENGTH';
				ELSIF(ArUser.ERR.No = ERR_RENAME_CURRENT_USER) THEN
					ArUser.ERR.Text := 'ERR: Can not rename user that is logged in';
				ELSE
					ArUser.ERR.Text := 'Error executing command';
				END_IF
				// Make sure we dont exceed maximum number of web clients
				IF(ArUser.PAR.VisuSlotID < SIZEOF(ArUser.VIS)/SIZEOF(ArUser.VIS[0])) THEN
					ArUser.VIS[ArUser.PAR.VisuSlotID].ShowMessageBoxError := TRUE;
				END_IF
				// --------------------------------------------------------------------------------------------------------------------
				// Return to idle state
				IF ArUser.CMD.ErrorReset THEN
					UserCounter := 1;
					RoleCounter := 0;

					brsmemset(ADR(ArUser.ERR), 0, SIZEOF(ArUser.ERR));
					ArUser.CMD.ErrorReset := FALSE;
					ArUser.VIS[ArUser.PAR.VisuSlotID].ShowMessageBoxError := FALSE;
					UserManagementState := IdleUser;
				END_IF;
				brsmemset(ADR(ArUser.CMD), 0, SIZEOF(ArUser.CMD));
				RETURN;
		END_CASE;
	END_FOR;

END_PROGRAM
```
